FUNCTION_BLOCK FB_ROOM IMPLEMENTS I_Room
VAR
	// Array of registered lamps
	iLamps 		: ARRAY[Param.INDEX_START..Param.MAX_LAMPS] OF I_Lamp;
END_VAR

METHOD AddLamp : BOOL
VAR_INPUT
	(* Lamp interface*)
	iLamp	: I_Lamp;
END_VAR

VAR
	// Loop Counter
	nIndex	: INT;
END_VAR
AddLamp := FALSE;
// Check to see if the reference is valid, if not return immediately
IF (iLamp = 0) THEN
	RETURN;
END_IF

// Is the lamp already registered?
FOR nIndex := Param.INDEX_START TO Param.MAX_LAMPS DO
	IF (THIS^.iLamps[nIndex] = iLamp) THEN
		AddLamp := TRUE;
		RETURN;
	END_IF
END_FOR

// Save it to the array if it's not
FOR nIndex := Param.INDEX_START TO  Param.MAX_LAMPS DO
	IF (THIS^.iLamps[nIndex] = 0) THEN
		THIS^.iLamps[nIndex] := iLamp;
		AddLamp := TRUE;
		EXIT;					
	END_IF
END_FOR
END_METHOD

METHOD Control : BOOL
VAR_INPUT
	(* Motion Sensor for the room*)
	bMotionSensor	: BOOL;
END_VAR

VAR
	nIndex: INT;
END_VAR
Control := FALSE;
FOR nIndex := Param.INDEX_START TO  Param.MAX_LAMPS DO
	IF bMotionSensor AND (THIS^.iLamps[nIndex] <> 0) THEN
		iLamps[nIndex].ON();
		Control := TRUE;
	ELSIF (THIS^.iLamps[nIndex] <> 0) THEN
		iLamps[nIndex].OFF();
	END_IF
END_FOR
END_METHOD

METHOD FB_exit : BOOL
VAR_INPUT
	bInCopyCode : BOOL; // if TRUE, the exit method is called for exiting an instance that is copied afterwards (online change).
END_VAR

VAR
	nIndex: INT;
END_VAR
FOR nIndex := 1 TO Param.MAX_LAMPS DO
	iLamps[nIndex] := 16#00;
END_FOR
END_METHOD

METHOD RemoveLamp : BOOL
VAR_INPUT
	(* Lamp interface*)
	iLamp	: I_Lamp;
END_VAR

VAR
	// Loop Counter
	nIndex	: INT;
END_VAR
RemoveLamp := FALSE;

IF (iLamp = 0) THEN
	RETURN;
END_IF

FOR nIndex := Param.INDEX_START TO  Param.MAX_LAMPS DO
	IF (THIS^.iLamps[nIndex] = iLamp) THEN
		THIS^.iLamps[nIndex] := 0;
		RemoveLamp := TRUE;	
	END_IF
END_FOR
END_METHOD

END_FUNCTION_BLOCK

(* stored: Version 1.1.0.1, ProductVersion 3.1.4024.6
   POU FB_ROOM: Id {5730381b-b9c1-4611-ba78-d6de9c2f1745}, SpecialFunc None
   Method AddLamp: Id {f3f5ec88-9fa8-443f-a1eb-ca1df337bdeb}
   Method Control: Id {4a4abe04-5f89-4572-8019-2240322cfc88}
   Method FB_exit: Id {dc28739e-820d-4233-a94e-5d153f890934}
   Method RemoveLamp: Id {28099617-1ec8-42cb-8f5b-89a6d4ec2c8b} *)
